PROGRAM TestRealPower
VAR
	currentCycle: INT := 0;
	cycleCount: INT := 0;
	switch: BOOL := FALSE;
END_VAR

IF currentCycle < GVL.cyclesToSkip THEN
	currentCycle := currentCycle + 1;
	RETURN; // Skip cycle
ELSE
	currentCycle := 0;
END_IF

cycleCount := cycleCount + 1;
GVL.arControllerData[GVL.currentIndex] := GVL.iHeaterActuator;
GVL.arTempData[GVL.currentIndex] := GVL.rTempSensor;
GVL.arRealPowerData[GVL.currentIndex] := GVL.iRealPower;
GVL.currentIndex := GVL.currentIndex + 1;

IF NOT switch AND GVL.iHeaterActuator = 100 THEN
	switch := TRUE;
END_IF

IF cycleCount MOD 100 = 0 THEN
	IF switch THEN
		GVL.iHeaterActuator := GVL.iHeaterActuator - 50;
	ELSE
		GVL.iHeaterActuator := GVL.iHeaterActuator + 50;
	END_IF

END_IF

END_PROGRAM

(* stored: Version 1.1.0.1, ProductVersion 3.1.4024.12
   POU TestRealPower: Id {644be3b1-3417-46ce-ab64-24cf25ee5f25}, SpecialFunc None *)
